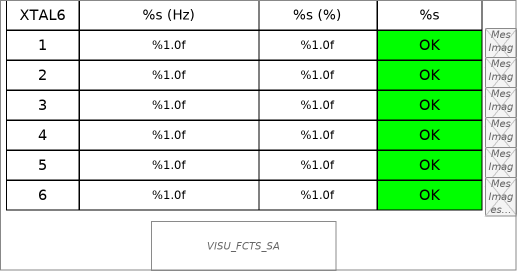
VISUALIZATION VISU_XTAL6_PROD  // 517x271, background image fond_blanc_1280_1024
VAR_IN_OUT
	m_Input_XTAL6 : BLOCK_XTAL6;
END_VAR
    RoundedRectangle (258,30 119x30), "%1.0f", text variable: m_Input_XTAL6.STATE_LIFE[1]
    RoundedRectangle (258,60 119x30), "%1.0f", text variable: m_Input_XTAL6.STATE_LIFE[2]
    RoundedRectangle (258,90 119x30), "%1.0f", text variable: m_Input_XTAL6.STATE_LIFE[3]
    RoundedRectangle (6,30 73x30), "1"
    RoundedRectangle (6,60 73x30), "2"
    RoundedRectangle (6,90 73x30), "3"
    RoundedRectangle (258,0 119x30), "%s (%)", text list: 'TextList_IC6', text index: 13
    RoundedRectangle (377,0 105x30), "%s", text list: 'TextList_IC6', text index: 14
    RoundedRectangle (377,30 105x30), "FAIL", invisible if: NOT m_Input_XTAL6.STATE_QF1
    RoundedRectangle (377,30 105x30), "OK", invisible if: (m_Input_XTAL6.STATE_QF1) <> 0
    RoundedRectangle (377,60 105x30), "FAIL", invisible if: NOT m_Input_XTAL6.STATE_QF2
    RoundedRectangle (377,60 105x30), "OK", invisible if: (m_Input_XTAL6.STATE_QF2) <> 0
    RoundedRectangle (377,90 105x30), "FAIL", invisible if: NOT m_Input_XTAL6.STATE_QF3
    RoundedRectangle (377,90 105x30), "OK", invisible if: (m_Input_XTAL6.STATE_QF3) <> 0
    RoundedRectangle (258,120 119x30), "%1.0f", text variable: m_Input_XTAL6.STATE_LIFE[4]
    RoundedRectangle (258,150 119x30), "%1.0f", text variable: m_Input_XTAL6.STATE_LIFE[5]
    RoundedRectangle (258,180 119x30), "%1.0f", text variable: m_Input_XTAL6.STATE_LIFE[6]
    RoundedRectangle (6,120 73x30), "4"
    RoundedRectangle (6,150 73x30), "5"
    RoundedRectangle (6,180 73x30), "6"
    RoundedRectangle (377,120 105x30), "FAIL", invisible if: NOT m_Input_XTAL6.STATE_QF4
    RoundedRectangle (377,120 105x30), "OK", invisible if: (m_Input_XTAL6.STATE_QF4) <> 0
    RoundedRectangle (377,150 105x30), "FAIL", invisible if: NOT m_Input_XTAL6.STATE_QF5
    RoundedRectangle (377,150 105x30), "OK", invisible if: (m_Input_XTAL6.STATE_QF5) <> 0
    RoundedRectangle (377,180 105x30), "FAIL", invisible if: NOT m_Input_XTAL6.STATE_QF6
    RoundedRectangle (377,180 105x30), "OK", invisible if: (m_Input_XTAL6.STATE_QF6) <> 0
    RoundedRectangle (6,0 73x30), "XTAL6"
    RoundedRectangle (79,30 180x30), "%1.0f", text variable: m_Input_XTAL6.STATE_FREQUENCY[1]
    RoundedRectangle (79,60 180x30), "%1.0f", text variable: m_Input_XTAL6.STATE_FREQUENCY[2]
    RoundedRectangle (79,90 180x30), "%1.0f", text variable: m_Input_XTAL6.STATE_FREQUENCY[3]
    RoundedRectangle (79,0 180x30), "%s (Hz)", text list: 'TextList_IC6', text index: 12
    RoundedRectangle (79,120 180x30), "%1.0f", text variable: m_Input_XTAL6.STATE_FREQUENCY[4]
    RoundedRectangle (79,150 180x30), "%1.0f", text variable: m_Input_XTAL6.STATE_FREQUENCY[5]
    RoundedRectangle (79,180 180x30), "%1.0f", text variable: m_Input_XTAL6.STATE_FREQUENCY[6]
    Image (485,28 32x39), invisible if: NOT m_Input_XTAL6.ALM_SURV_ACTIVITY_QZ1.DEF AND NOT m_Input_XTAL6.ALM_SURV_LIFE_QZ1.DEF, image: MesImages.warning
    Image (485,57 32x39), invisible if: NOT m_Input_XTAL6.ALM_SURV_ACTIVITY_QZ2.DEF AND NOT m_Input_XTAL6.ALM_SURV_LIFE_QZ2.DEF, image: MesImages.warning
    Image (485,87 32x39), invisible if: NOT m_Input_XTAL6.ALM_SURV_ACTIVITY_QZ3.DEF AND NOT m_Input_XTAL6.ALM_SURV_LIFE_QZ3.DEF, image: MesImages.warning
    Image (485,117 32x39), invisible if: NOT m_Input_XTAL6.ALM_SURV_ACTIVITY_QZ4.DEF AND NOT m_Input_XTAL6.ALM_SURV_LIFE_QZ4.DEF, image: MesImages.warning
    Image (485,147 32x39), invisible if: NOT m_Input_XTAL6.ALM_SURV_ACTIVITY_QZ5.DEF AND NOT m_Input_XTAL6.ALM_SURV_LIFE_QZ5.DEF, image: MesImages.warning
    Image (485,177 32x39), invisible if: NOT m_Input_XTAL6.ALM_SURV_ACTIVITY_QZ6.DEF AND NOT m_Input_XTAL6.ALM_SURV_LIFE_QZ6.DEF, image: MesImages.warning
    Frame (151,221 185x50)
        shows VISU_FCTS_SA(m_Input_ID_XML := 21, m_Input_Operation := m_Input_XTAL6.OP_Scan_Quartz, m_Input_UserRight := PRG_USER.ACTU_USER.FONCTION_SA AND NOT MACHINE.STATE_PROD)
END_VISUALIZATION

(* stored: Version 1.1.0.1, ProductVersion 3.1.4024.12
   Visu VISU_XTAL6_PROD: Id {88ae19af-d8e1-4f8b-be41-edaf234dec36} *)
